// TIA Portal V20 export
TYPE "typeCmControlNodeInterlock"
// stored: Namespace Unit1.Em12
   STRUCT
      stackNgBoxLoading : "LER_typeTwoWayActuatorInterlock";
      stackNgBoxUnitMover : "LER_typeTwoWayActuatorInterlock";
      stackNgBoxClampLeft : "LER_typeTwoWayActuatorInterlock";
      stackNgBoxClampRight : "LER_typeTwoWayActuatorInterlock";
      stackNgBoxClampMover : "LER_typeTwoWayActuatorInterlock";
      stackNgBoxLift : "LER_typeTwoWayActuatorInterlock";
      stackNgBoxLock : "LER_typeTwoWayActuatorInterlock";
   END_STRUCT;
END_TYPE
